Xinje XDPPro project, PLC1: XDH-60T4 (software 3.7.14b 2022-06-24)

PROGRAM 梯形图

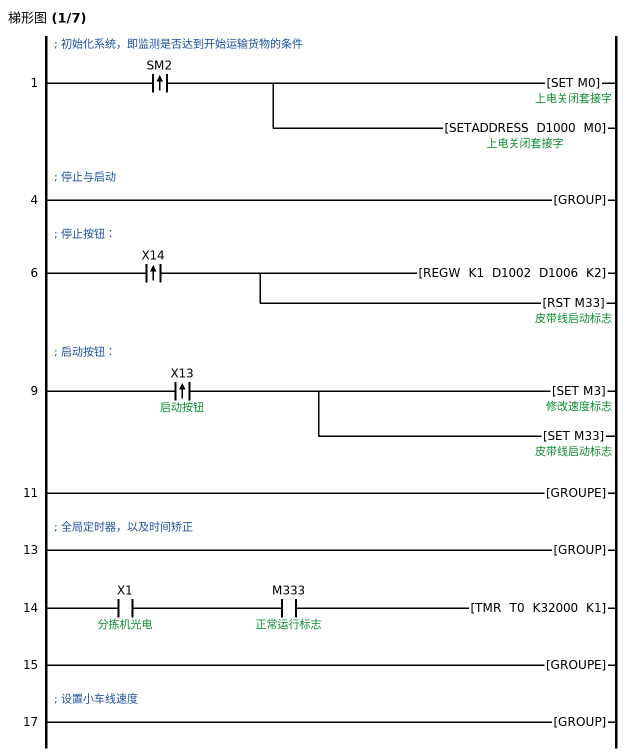
; 初始化系统，即监测是否达到开始运输货物的条件
LDP    SM2
SET    M0	; 上电关闭套接字
SETADDRESS D1000 M0	; 上电关闭套接字
; 停止与启动
GROUP
; 停止按钮：
LDP    X14
REGW   K1 D1002 D1006 K2
RST    M33	; 皮带线启动标志
; 启动按钮：
LDP    X13	; 启动按钮
SET    M3	; 修改速度标志
SET    M33	; 皮带线启动标志
GROUPE
; 全局定时器，以及时间矫正
GROUP
LD     X1	; 分拣机光电
AND    M333	; 正常运行标志
TMR    T0 K32000 K1
GROUPE
; 设置小车线速度
GROUP

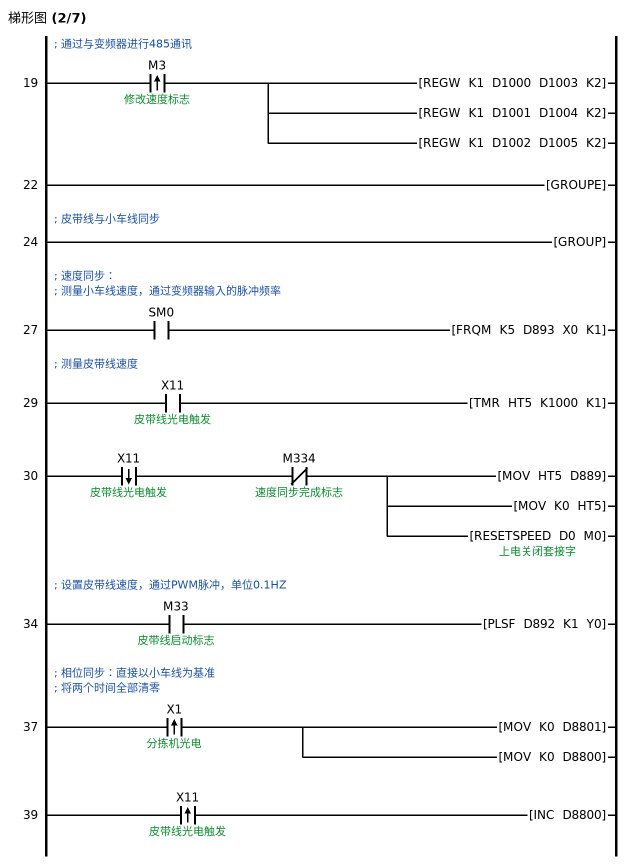
; 通过与变频器进行485通讯
LDP    M3	; 修改速度标志
REGW   K1 D1000 D1003 K2
REGW   K1 D1001 D1004 K2
REGW   K1 D1002 D1005 K2
GROUPE
; 皮带线与小车线同步
GROUP
; 速度同步：
; 测量小车线速度，通过变频器输入的脉冲频率
LD     SM0
FRQM   K5 D893 X0 K1
; 测量皮带线速度
LD     X11	; 皮带线光电触发
TMR    HT5 K1000 K1
LDF    X11	; 皮带线光电触发
ANI    M334	; 速度同步完成标志
MOV    HT5 D889
MOV    K0 HT5
RESETSPEED D0 M0	; 上电关闭套接字
; 设置皮带线速度，通过PWM脉冲，单位0.1HZ
LD     M33	; 皮带线启动标志
PLSF   D892 K1 Y0
; 相位同步：直接以小车线为基准
; 将两个时间全部清零
LDP    X1	; 分拣机光电
MOV    K0 D8801
MOV    K0 D8800
LDP    X11	; 皮带线光电触发
INC    D8800

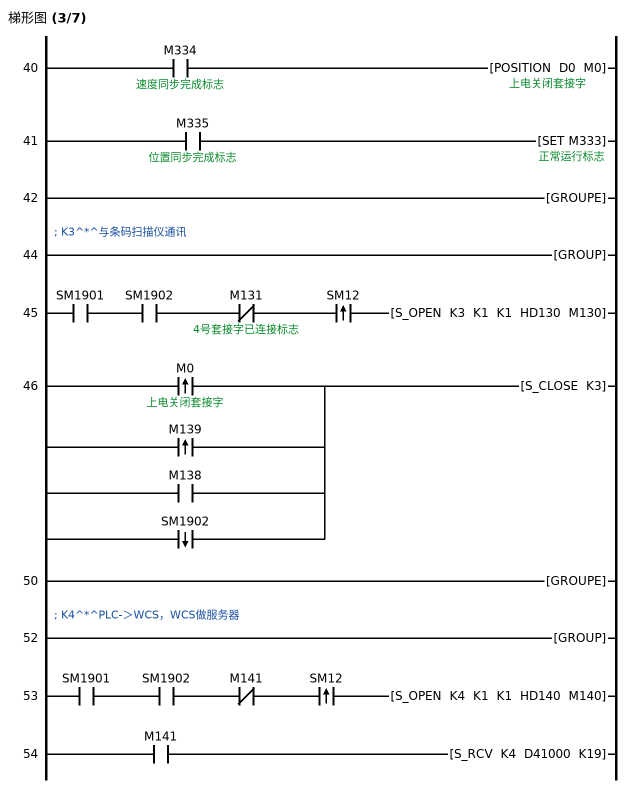
LD     M334	; 速度同步完成标志
POSITION D0 M0	; 上电关闭套接字
LD     M335	; 位置同步完成标志
SET    M333	; 正常运行标志
GROUPE
; K3^*^与条码扫描仪通讯
GROUP
LD     SM1901
AND    SM1902
ANI    M131	; 4号套接字已连接标志
ANDP   SM12
S_OPEN K3 K1 K1 HD130 M130
LDP    M0	; 上电关闭套接字
ORP    M139
OR     M138
ORF    SM1902
S_CLOSE K3
GROUPE
; K4^*^PLC-＞WCS，WCS做服务器
GROUP
LD     SM1901
AND    SM1902
ANI    M141
ANDP   SM12
S_OPEN K4 K1 K1 HD140 M140
LD     M141
S_RCV  K4 D41000 K19

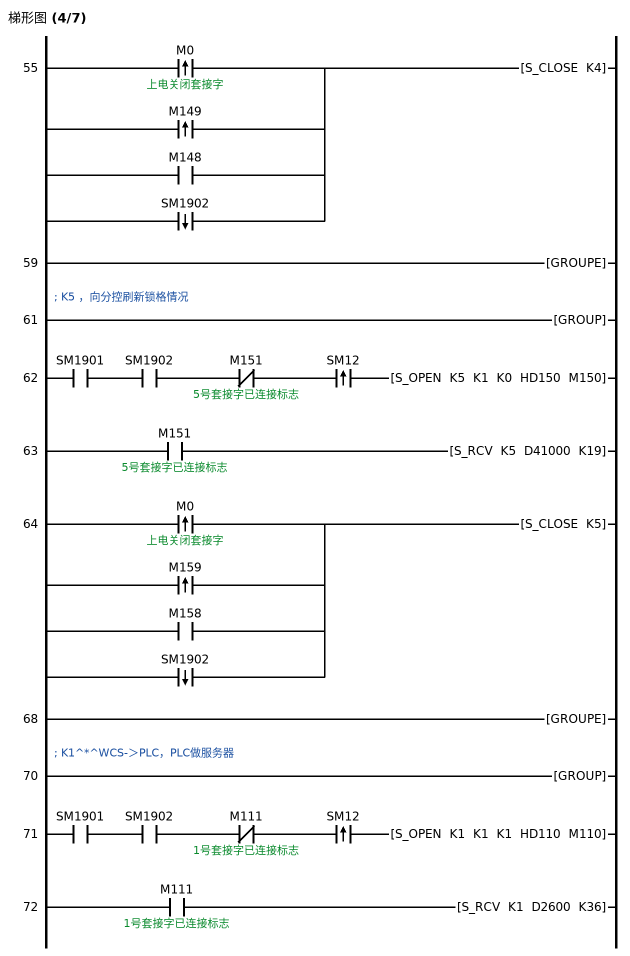
LDP    M0	; 上电关闭套接字
ORP    M149
OR     M148
ORF    SM1902
S_CLOSE K4
GROUPE
; K5 ，向分控刷新锁格情况
GROUP
LD     SM1901
AND    SM1902
ANI    M151	; 5号套接字已连接标志
ANDP   SM12
S_OPEN K5 K1 K0 HD150 M150
LD     M151	; 5号套接字已连接标志
S_RCV  K5 D41000 K19
LDP    M0	; 上电关闭套接字
ORP    M159
OR     M158
ORF    SM1902
S_CLOSE K5
GROUPE
; K1^*^WCS-＞PLC，PLC做服务器
GROUP
LD     SM1901
AND    SM1902
ANI    M111	; 1号套接字已连接标志
ANDP   SM12
S_OPEN K1 K1 K1 HD110 M110
LD     M111	; 1号套接字已连接标志
S_RCV  K1 D2600 K36

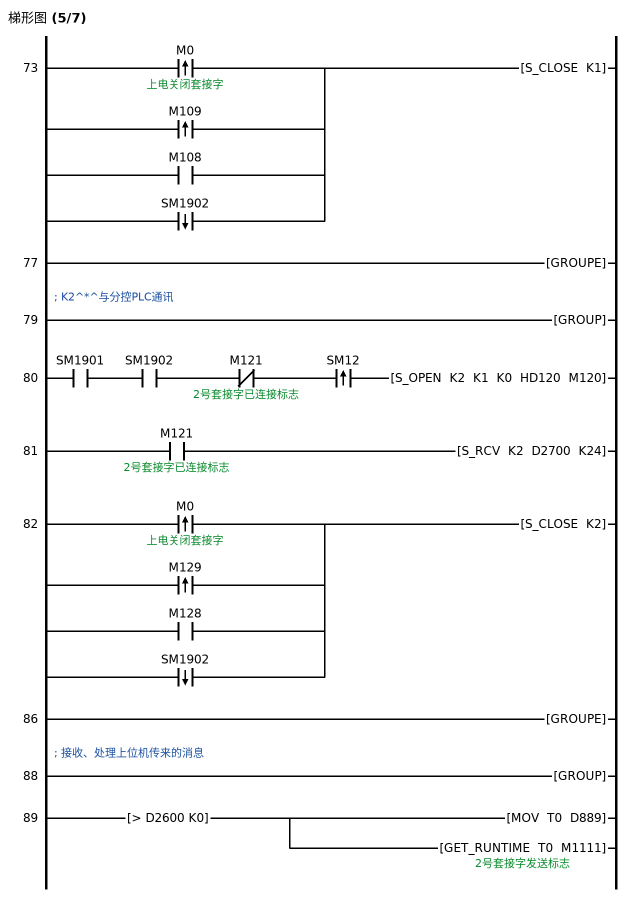
LDP    M0	; 上电关闭套接字
ORP    M109
OR     M108
ORF    SM1902
S_CLOSE K1
GROUPE
; K2^*^与分控PLC通讯
GROUP
LD     SM1901
AND    SM1902
ANI    M121	; 2号套接字已连接标志
ANDP   SM12
S_OPEN K2 K1 K0 HD120 M120
LD     M121	; 2号套接字已连接标志
S_RCV  K2 D2700 K24
LDP    M0	; 上电关闭套接字
ORP    M129
OR     M128
ORF    SM1902
S_CLOSE K2
GROUPE
; 接收、处理上位机传来的消息
GROUP
LD>    D2600 K0
MOV    T0 D889
GET_RUNTIME T0 M1111	; 2号套接字发送标志

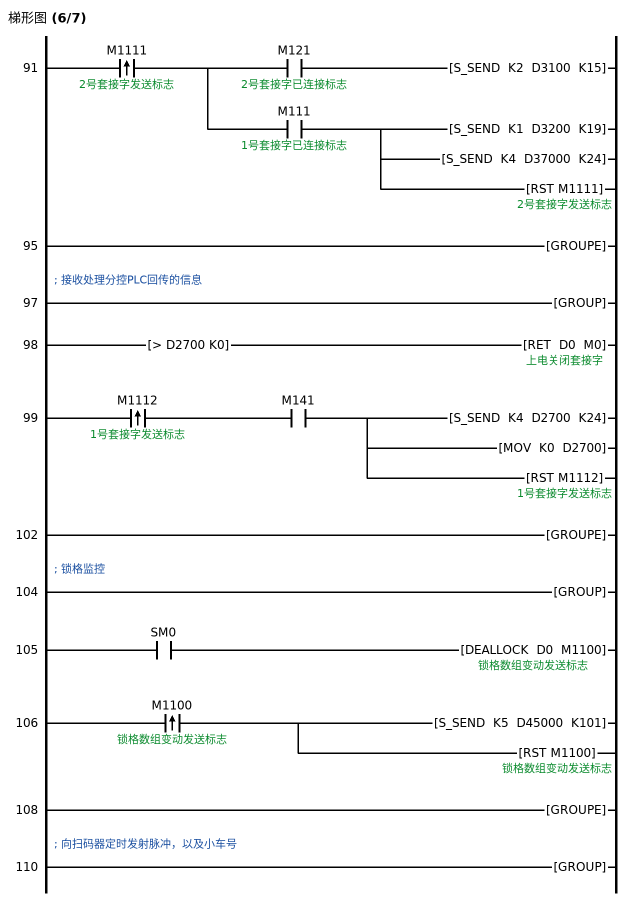
LDP    M1111	; 2号套接字发送标志
MPS
AND    M121	; 2号套接字已连接标志
S_SEND K2 D3100 K15
MPP
AND    M111	; 1号套接字已连接标志
S_SEND K1 D3200 K19
S_SEND K4 D37000 K24
RST    M1111	; 2号套接字发送标志
GROUPE
; 接收处理分控PLC回传的信息
GROUP
LD>    D2700 K0
RET    D0 M0	; 上电关闭套接字
LDP    M1112	; 1号套接字发送标志
AND    M141
S_SEND K4 D2700 K24
MOV    K0 D2700
RST    M1112	; 1号套接字发送标志
GROUPE
; 锁格监控
GROUP
LD     SM0
DEALLOCK D0 M1100	; 锁格数组变动发送标志
LDP    M1100	; 锁格数组变动发送标志
S_SEND K5 D45000 K101
RST    M1100	; 锁格数组变动发送标志
GROUPE
; 向扫码器定时发射脉冲，以及小车号
GROUP

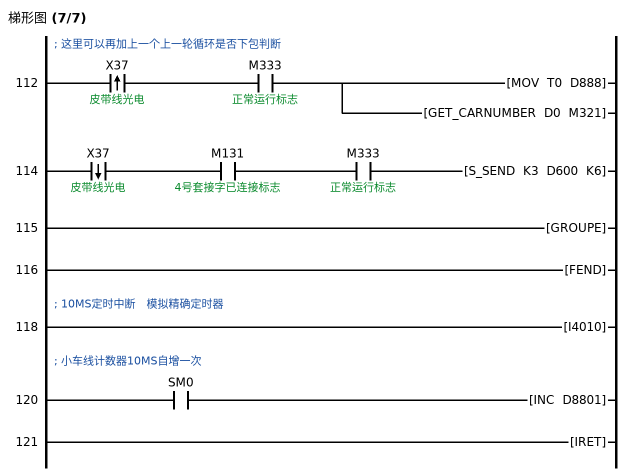
; 这里可以再加上一个上一轮循环是否下包判断
LDP    X37	; 皮带线光电
AND    M333	; 正常运行标志
MOV    T0 D888
GET_CARNUMBER D0 M321
LDF    X37	; 皮带线光电
AND    M131	; 4号套接字已连接标志
AND    M333	; 正常运行标志
S_SEND K3 D600 K6
GROUPE
FEND
; 10MS定时中断　模拟精确定时器
I4010
; 小车线计数器10MS自增一次
LD     SM0
INC    D8801
IRET

COMMENTS (devices not used above)
M101	1号套接字已连接
M99	3号套接字发送标志
HD10	定时器最大值
HD11	定时器数量
Y1	控制伺服电机方向

C FUNCTION BLOCK deallock.fcb
/* 处理、检测锁格的情况
#EXPORT_ENTRY_BEGIN(DEALLOCK)
//    类型              模式             个数               映射          注释
W = { type = "PINT16S", mode = [In,Out], count = "unknown", map = [D,HD], comment = "" }
B = { type = "BIT"    , mode = [In,Out], count = "unknown", map = [M,HM], comment = "" }
#EXPORT_ENTRY_END */
/*************************************************************************
 * FunctionBlockName:  DEALLOCK
 * Version:            1.0.0
 * Author:             rpl
 * UpdateTime:         2022-09-13 14:35:26
 * Comment:            处理、检测锁格的情况
**************************************************************************/

/**
 * @summary 
 * @param W 
 * @param B 
 */
 
 #include"func1.h"

void DEALLOCK(PINT16S W,BIT B)
{
	#define SysRegAddr_HD_D_HM_M_X_Y
	
    *(LOCKFIRSTADDRESS) = 0x02;
	for(int i = 30; i<=SIZEOFLATTICE;i++)
    {
    	if(X[i]!= *(LOCKFIRSTADDRESS+i+1))
        {
                //发送位置1
                M[1100] = 1;
        }
        * ( LOCKFIRSTADDRESS + i+1 ) = X[i];
    }
    return;
}

C FUNCTION BLOCK dealwith_k1.fcb
/* #EXPORT_ENTRY_BEGIN(DEALWITH_K1)
//    类型              模式             个数               映射          注释
W = { type = "PINT16S", mode = [In,Out], count = "unknown", map = [D,HD], comment = "" }
B = { type = "BIT"    , mode = [In,Out], count = "unknown", map = [M,HM], comment = "" }
#EXPORT_ENTRY_END */
/*************************************************************************
 * FunctionBlockName:  DEALWITH_K1
 * Version:            1.0.0
 * Author:             
 * UpdateTime:         2022-08-22 14:10:12
 * Comment:            
**************************************************************************/

/**
 * @summary 
 * @param W 
 * @param B 
 */
void DEALWITH_K1(PINT16S W,BIT B)
{
	#define SysRegAddr_HD_D_HM_M
    M[103] = 0;
    M[1112]　 = 0;

}

C FUNCTION BLOCK dealwith_k2.fcb
/* #EXPORT_ENTRY_BEGIN(DEALWITH_K2)
//    类型              模式             个数               映射          注释
W = { type = "PINT16S", mode = [In,Out], count = "unknown", map = [D,HD], comment = "" }
B = { type = "BIT"    , mode = [In,Out], count = "unknown", map = [M,HM], comment = "" }
#EXPORT_ENTRY_END */
/*************************************************************************
 * FunctionBlockName:  DEALWITH_K2
 * Version:            1.0.0
 * Author:             
 * UpdateTime:         2022-08-22 14:08:06
 * Comment:            
**************************************************************************/

/**
 * @summary 
 * @param W 
 * @param B 
 */
void DEALWITH_K2(PINT16S W,BIT B)
{
	#define SysRegAddr_HD_D_HM_M
    M[113] = 0;
    M[1111] = 0;

}

C FUNCTION BLOCK func1.fcb
/* #EXPORT_ENTRY_BEGIN(FUNC1)
//    类型              模式             个数               映射          注释
W = { type = "PINT16S", mode = [In,Out], count = "unknown", map = [D,HD], comment = "" }
B = { type = "BIT"    , mode = [In,Out], count = "unknown", map = [M,HM], comment = "" }
#EXPORT_ENTRY_END */
/*************************************************************************
 * FunctionBlockName:  FUNC1
 * Version:            1.0.0
 * Author:             
 * UpdateTime:         2022-08-18 08:24:01
 * Comment:            
**************************************************************************/

/**
 * @summary 
 * @param W 
 * @param B 
 */
void FUNC1(PINT16S W,BIT B)
{
	#define SysRegAddr_HD_D_HM_M

}

C FUNCTION BLOCK get_carnumber.fcb
/* 输入时间，返回当前相机拍摄的小车号
#EXPORT_ENTRY_BEGIN(GET_CARNUMBER)
//    类型              模式             个数               映射          注释
W = { type = "PINT16S", mode = [In,Out], count = "unknown", map = [D,HD], comment = "" }
B = { type = "BIT"    , mode = [In,Out], count = "unknown", map = [M,HM], comment = "" }
#EXPORT_ENTRY_END */
/*************************************************************************
 * FunctionBlockName:  GET_CARNUMBER
 * Version:            1.0.0
 * Author:             rpl
 * UpdateTime:         2022-08-10 14:44:36
 * Comment:            输入时间,返回当前相机拍摄的小车号,将返回数据处理发给扫码仪
**************************************************************************/

/**
 * @summary
 * @param W
 * @param B
 */
#include"func1.h"


void GET_CARNUMBER ( PINT16S W, BIT B )
{
#define SysRegAddr_HD_D_HM_M_T
    /*根据时间判断出当前是多少号小车(小车从0号开始排序) */
    INT32U tmpp =  Speed * PassedTime*10;
    INT16U carnumber;
    if(tmpp >= Light2CameraPosition)
    {
        carnumber = ( (tmpp -Light2CameraPosition) / DistanceOfCar ) + 1;  //判断是哪个小车,用来绑定小车的控制电机计时时间
    }
    else{
        carnumber = ( (tmpp + Camera_Position)/ DistanceOfCar ) + 1;  //判断是哪个小车,用来绑定小车的控制电机计时时间
        
    }
    



    /***将小车号数据写入寄存器,起始位置D600,6个***/
    //消息头
    //int TempCar = carnumber;
    * ( SendToCameraFirstAddress ) = 0x02;
    //千位
    * ( SendToCameraFirstAddress + 1 ) = 0x30;
    //百位
    * ( SendToCameraFirstAddress + 2 ) = 48 + ( carnumber / 100 ) % 10 ;
    //十位
    * ( SendToCameraFirstAddress + 3 ) = 48 + ( carnumber / 10 ) % 10;
    //个位
    * ( SendToCameraFirstAddress + 4 ) = 48 + carnumber % 10;
    //结束符
    * ( SendToCameraFirstAddress + 5 ) = 0x03;



    //M[321] = 1;
    return;
}

C FUNCTION BLOCK get_runtime.fcb
/* D[100]返回某个电机在多少秒后运行,D[101]返回判断出的小车号，以此来进行绑定
#EXPORT_ENTRY_BEGIN(GET_RUNTIME)
//    类型          模式             个数               映射          注释
w = { type = "BIT", mode = [In]    , count = "1"      , map = [T]   , comment = "时间差" }
B = { type = "BIT", mode = [In,Out], count = "unknown", map = [M,HM], comment = ""    }
#EXPORT_ENTRY_END */
/*************************************************************************
 * FunctionBlockName:  GET_RUNTIME
 * Version:            1.0.0
 * Author:             rpl
 * UpdateTime:         2022-07-25 16:38:06
 * Comment:            处理上位机发来的数据，返回的ACK报文，写入发送缓冲区，
**************************************************************************/

/**
 * @summary
 * @param w 时间差
 * @param B
 */
#include "func1.h"

void GET_RUNTIME ( BIT w, BIT B )
{
#define SysRegAddr_HD_D_HM_M_T
    /** 分拣指令	0x02(起始符(16进制))	1(报文类型ASCII)
        齐格控制	0x02(起始符(16进制))	2(报文类型ASCII)
        锁格控制	0x02(起始符(16进制))	3(报文类型ASCII)
    */


    int master = * ( RCVDateFirstAddress + 1 );
    switch ( master )
    {
        case 49:
        {
            /**先处理接受到的报文,得到其中的小车号,格口号**/
            //先处理小车号码
            INT16U Car_Mark ;
            Car_Mark = ( *(RCVDateFirstAddress+10) - 48 ) * 1000 + ( *(RCVDateFirstAddress+11) - 48 ) * 100 + ( *(RCVDateFirstAddress+12) - 48 ) * 10 + *(RCVDateFirstAddress+13) - 48 ;
            
            INT16U Bourn1, Bourn2, Bourn3, Bourn4;
            INT16U  NeedTime1, NeedTime2, NeedTime3, NeedTime4;
            //如果小车号为0,即为返回报文 ,暂时不作处理直接丢弃
            if ( Car_Mark == 0 )
            {
                return;
            }
            //处理格口号
            Bourn1 = ( *(RCVDateFirstAddress+14) - 48 ) * 1000 + ( *(RCVDateFirstAddress+15) - 48 ) * 100 + ( *(RCVDateFirstAddress+16) - 48 ) * 10 + *(RCVDateFirstAddress+17) - 48 ;
            Bourn2 = ( *(RCVDateFirstAddress+18) - 48 ) * 1000 + ( *(RCVDateFirstAddress+19) - 48 ) * 100 + ( *(RCVDateFirstAddress+20) - 48 ) * 10 + *(RCVDateFirstAddress+21) - 48 ;
            Bourn3 = ( *(RCVDateFirstAddress+22) - 48 ) * 1000 + ( *(RCVDateFirstAddress+23) - 48 ) * 100 + ( *(RCVDateFirstAddress+24) - 48 ) * 10 + *(RCVDateFirstAddress+25) - 48 ;
            Bourn4 = ( *(RCVDateFirstAddress+26) - 48 ) * 1000 + ( *(RCVDateFirstAddress+27) - 48 ) * 100 + ( *(RCVDateFirstAddress+28) - 48 ) * 10 + *(RCVDateFirstAddress+29) - 48 ;
            INT16U time = D[889] * 10;
            NeedTime1 = ( Bourn1 * DistanceOfCut + ( Car_Mark - 1 ) * DistanceOfCar ) / Speed  - time; //总时间减去已经用的时间
            NeedTime2 = ( Bourn2 * DistanceOfCut + ( Car_Mark - 1 ) * DistanceOfCar ) / Speed  - time;
            NeedTime3 = ( Bourn3 * DistanceOfCut + ( Car_Mark - 1 ) * DistanceOfCar ) / Speed  - time;
            NeedTime4 = ( Bourn4 * DistanceOfCut + ( Car_Mark - 1 ) * DistanceOfCar ) / Speed  - time;
            //}
            
            //将数据填入发送缓冲区
            //首位
            * ( SendToLowPLCBuffAddress ) = 0x02;
            //定时1
            * ( SendToLowPLCBuffAddress + 1 ) = NeedTime1 >> 8;
            * ( SendToLowPLCBuffAddress + 2 ) = ( NeedTime1 << 8 ) >> 8;
            //定时2
            * ( SendToLowPLCBuffAddress + 3 ) = NeedTime2 >> 8;
            * ( SendToLowPLCBuffAddress + 4 ) = ( NeedTime2 << 8 ) >> 8;
            //定时3
            * ( SendToLowPLCBuffAddress + 5 ) = NeedTime3 >> 8;
            * ( SendToLowPLCBuffAddress + 6 ) = ( NeedTime3 << 8 ) >> 8;
            //定时四
            * ( SendToLowPLCBuffAddress + 7 ) = NeedTime4 >> 8;
            * ( SendToLowPLCBuffAddress + 8 ) = ( NeedTime4 << 8 ) >> 8;
            //格口
            
            //格口1
            * ( SendToLowPLCBuffAddress + 9 ) = Bourn1;
            //格口2
            * ( SendToLowPLCBuffAddress + 10 ) = Bourn2;
            //格口3
            * ( SendToLowPLCBuffAddress + 11 ) = Bourn3;
            //格口4
            * ( SendToLowPLCBuffAddress + 12 ) = Bourn4;
            //小车号
            * ( SendToLowPLCBuffAddress + 13 ) = Car_Mark;
            //命令语
            * ( SendToLowPLCBuffAddress + 14 ) = master;
            break;
        }
        case 50: //齐格指令
        break;
        case 51://锁格指令
        break;
    }
    
    
    



    /**************************************处理向上位机回复ACK信息************************
     1.起始位置D3200               ***
     2.发送19个寄存器的数据        ***
     *************/
     *(SendACKToWCSFiestAddress) = 0x02;

    /**将报文编号复制到1号套接字发送缓冲区*/
    for ( int i = 1; i <= 8; i++ )
    {
        *(SendACKToWCSFiestAddress +i) = *(RCVDateFirstAddress+1+i);
    }
    for ( int i = 9; i <= 12; i++ )
    {
        *(SendACKToWCSFiestAddress +i)  = 48;
    }

    for ( int i = 13; i <= 17; i++ )
    {
        *(SendACKToWCSFiestAddress +i) = 0x20;
    }
    //结束符
    *(SendACKToWCSFiestAddress +18) = 0x03;

    //将接受区的数据清零
    *(RCVDateFirstAddress) = 0;
    //出发发送数据用
    M[1111] = 1;
    return;
}

C FILE func1.h
#ifndef	_FUNC1_H
#define	_FUNC1_H
/*********宏定义用来存放需要的返回值************/
 //#define NEEDTIME D[3100]       //保存返回值
 //#define CAR      D[3102]        //存储判断出来的小车号
 //#define Bourn     D[3103]       //目的格口
 //#define Time      D[300]           //时间基点定时器的计数值 
#define D_D	     *(INT32S*)&D


/**********首地址************/
#define SendToLowPLCBuffAddress D+3100 //发送给分控的发送缓冲区首地址,总计15个寄存器
#define RCVDateFirstAddress D+2600      //上位机发来的数据缓冲区首地址，总计36个寄存器
#define SendACKToWCSFiestAddress D+3200 //向上位机回复ACK报文的数据缓冲区首地址，总计19个寄存器
#define SendToCameraFirstAddress D+600  //发给相机，6个寄存器
#define RCVDateFormLOW          D+2700  //分控分拣完成返回，24个寄存器
#define LOCKFIRSTADDRESS D+45000        //锁格队列首地址,101个寄存器
#define CarDateFirstAddress D+3300      //存放已有任务的小车数组


/* 存放一些函数中需要的参数 
所有的距离单位为毫米，时间单位为毫秒
 */
 
 
 #define TrackLength  50000         //轨道的长度
 #define  Speed  1                  //小车速度1mm/ms
 #define DistanceOfCar  400         //小车的间距(单位为：毫米)
 #define TIMELOSS  5                //电机启动时间偏移量(单位为：毫秒)

 #define Time_Offset 　0            //时间偏移量，由于没有进行实验测试暂时设置为0,该值是用来计算小车上的电机转动所需要的时间

 #define DistanceOfCut  750         //此处割口的间距 ————割口的长度加上割口间的距离

 #define  Camera_Position  600      //扫码设备->光电的距离
 #define Light2CameraPosition (TrackLength-Camera_Position)  //光电->扫码设备的距离

 #define Time  0                    //距离时间基点的时间

 
 #define SIZEOFLATTICE 100      //格口个数


//小车线与皮带线用
#define PassedTime      D[888]
#define NowSpeed        D[890]         //皮带线当前速度
#define CarSpeed        D[891]         //小车线速度
#define PulseFrequency  D[892]   //皮带线脉冲频率
#define FinallyFrequency  D[894]    //皮带线最终脉冲频率
#define CarFrequency    D[893]   //小车线反馈脉冲频率
#define speedAddress     D[1000]  //Modbus转速地址
#define PowerAddress     D[1001]  //转矩地址
#define MasterAddress    D[1002]  //命令符地址
#define speedValue       D[1003]  //转速数值
#define PowerValue       D[1004]  //转矩数值
#define MasterValue      D[1005]  //命令符
#define StopMaster       D[1006]    //电机停止
#define CarIncConter   D[8801]  //小车线当前时间
#define PulseIncConter D[8800]  //皮带线当前计数值

#define CameraEnableTime D[894]     //相机使能定时时间
#define DZCL        D[8802]     //转一圈需要的脉冲数

#endif

C FUNCTION BLOCK init.fcb
/* 初始化需要的数组，结构体
#EXPORT_ENTRY_BEGIN(INIT)
//    类型              模式             个数               映射          注释
W = { type = "PINT16S", mode = [In,Out], count = "unknown", map = [D,HD], comment = "" }
B = { type = "BIT"    , mode = [In,Out], count = "unknown", map = [M,HM], comment = "" }
#EXPORT_ENTRY_END */
/*************************************************************************
 * FunctionBlockName:  INIT
 * Version:            1.0.0
 * Author:             rpl
 * UpdateTime:         2022-09-13 15:01:51
 * Comment:            初始化需要的数组，结构体
**************************************************************************/

/**
 * @summary 
 * @param W 
 * @param B 
 */
 #include"func1.h"
void INIT(PINT16S W,BIT B)
{
	#define SysRegAddr_HD_D_HM_M
	for(int i = 0;i<=SIZEOFLATTICE; i++)
    {
        * ( LOCKFIRSTADDRESS + i ) = 0;
    }
	
	

}

C FUNCTION BLOCK position.fcb
/* 位置矫正，皮带线与分拣机的相位矫正。
#EXPORT_ENTRY_BEGIN(POSITION)
//    类型              模式             个数               映射          注释
W = { type = "PINT16S", mode = [In,Out], count = "unknown", map = [D,HD], comment = "" }
B = { type = "BIT"    , mode = [In,Out], count = "unknown", map = [M,HM], comment = "" }
#EXPORT_ENTRY_END */
/*************************************************************************
 * FunctionBlockName:  POSITION
 * Version:            1.0.0
 * Author:             rpl
 * UpdateTime:         2022-09-28 16:15:44
 * Comment:            位置矫正，皮带线与分拣机的相位矫正。
                        这里默认已经进行过基本的速度矫正
**************************************************************************/

/**
 * @summary 
 * @param W 
 * @param B 
 */
 #include"func1.h"
void POSITION(PINT16S W,BIT B)
{
	#define SysRegAddr_HD_D_HM_M
    /*需要做的事情
    1.两条线的计数器时间之差： 分拣机的可以通过时间进行自增 保持精度与皮带线相同或者大十倍
    2.频率对应的关系变量
    3.微调是通过固定值加减还是通过速度公式去追及，在追及的时候速度什么时候降到与分拣机相同，在下一次的光电信号到来之前是无法判断当前相位差的
    4.速度与频率关系的对应公式！！！
    */
    /*新增控制部分需要的参数 
    1.直线电机的运行速度 V    1.0 mm/ms  1.0 m/s
    2.伺服电机的电子齿轮比 K 10000:10000  
    3.伺服电机旋转一圈的长度 C   440 mm    
    4.脉冲：距离 = 10000 ： 500
    5.脉冲频率 H
    6. 伺服电机速度（单位 mm/s） =
    
    7. 伺服电机当前频率 PulseFrequency
    8.两条线的计数值之差 CounterDifference
    9.单位步进值  UnitStepValue
    */
    //int CarIncCounter; //乘以10等于小车线当前走的时间
    //int PulseFrequency;     //间距除以速度等于皮带线当前走的时间
    //int UnitStepValue =  DZCL*10 *DistanceOfCar / 0.44;
    int CarDistance  =  CarIncCounter * 10 * Speed; //单位ms
    int BeltDistance =  PulseIncConter * DistanceOfCar; // 单位mm
    int DistanceDifference = CarDistance - BeltDistance; //两条线的相位差
    /**拟通过单位步进值来进行处理，但应该是行不通的*/
    /*每次增加1000个脉冲——0.1375m/s的速度去追及*/
    if(DistanceDifference >=0)
    { 
        PulseFrequency += 1000 ;
    }
    else if(DistanceDifference < 0)
    {
        PulseFrequency -= 1000; 
    }

    //相位矫正完成
    if(DistanceDifference >= -10 || DistanceDifference <= 10 )
    {
        //将速度重置为最终速度
        PulseFrequency = FinallyFrequency;
        
        M[335] = 1;     //相位同步完成标志
    }
    else
    {
    M[335] = 0;
    }

return;
}

C FUNCTION BLOCK resetspeed.fcb
/* 皮带线速度向小车线靠近
#EXPORT_ENTRY_BEGIN(RESETSPEED)
//    类型              模式             个数               映射          注释
W = { type = "PINT16S", mode = [In,Out], count = "unknown", map = [D,HD], comment = "" }
B = { type = "BIT"    , mode = [In,Out], count = "unknown", map = [M,HM], comment = "" }
#EXPORT_ENTRY_END */
/*************************************************************************
 * FunctionBlockName:  RESETSPEED
 * Version:            1.0.0
 * Author:             
 * UpdateTime:         2022-10-06 17:14:06
 * Comment:            皮带线速度向小车线靠近
**************************************************************************/

/**
 * @summary 
 * @param W 
 * @param B 
 */
 #include"func1.h"
 #define TimeValue D[889]
void RESETSPEED(PINT16S W,BIT B)
{
	#define SysRegAddr_HD_D_HM_M
    float deviation = 0.05; //允许误差
    NowSpeed =  DistanceOfCar / TimeValue;//单位 mm/ms
    CarSpeed = CarFrequency * 0.1; //单位m/s
    if (NowSpeed < CarSpeed)
    { 
        //此处假设1000个脉冲转一圈
        PulseFrequency = PulseFrequency + ( ( CarSpeed - NowSpeed ) *1000/137.5);
        //百分比*额度转速*减速比 = 实际转速
        //实际转速*0.44 = 线速度
        //调整后的频率= 当前频率+差值速度*100000  /0.44/减速比/额定转速
    }
    else if(NowSpeed > CarSpeed)
    {
        PulseFrequency = PulseFrequency - ( ( NowSpeed -CarSpeed) *1000/137.5);
    }
    //脉冲乘以减速比
    PulseFrequency = PulseFrequency * 16;
	//当速度达到允许误差时，速度同步完成标志置1
	if(NowSpeed == CarSpeed || NowSpeed - CarSpeed <=deviation ||  CarSpeed - NowSpeed <=deviation )
	{
	    //保存速度同步完成的频率
        PulseFrequency = FinallyFrequency;
        M[334] = 1;
	}
	////超过最大允许误差时，将速度同步完成标志置0
	//else
	//{
	    
	    //M[334] = 0;
	//}
    return;
}

C FUNCTION BLOCK ret.fcb
/* 向上位机返回ack
#EXPORT_ENTRY_BEGIN(RET)
//    类型              模式             个数               映射          注释
W = { type = "PINT16S", mode = [In,Out], count = "unknown", map = [D,HD], comment = "" }
B = { type = "BIT"    , mode = [In,Out], count = "unknown", map = [M,HM], comment = "" }
#EXPORT_ENTRY_END */
/*************************************************************************
 * FunctionBlockName:  RET
 * Version:            1.0.0
 * Author:             
 * UpdateTime:         2022-09-08 15:23:59
 * Comment:            向上位机返回ack
**************************************************************************/

/**
 * @summary 
 * @param W 
 * @param B 
 */
 #define SendToWCSFirstAddress D+37000
 #include"func1.h"
void RET(PINT16S W,BIT B)
{
	#define SysRegAddr_HD_D_HM_M
	//落格成功返回
	
	//起始符
    *(SendToWCSFirstAddress) = 0x02;
    //分拣完成
    *(SendToWCSFirstAddress+1) = 53;
    
    //报文编号
    for(int i = 2; i<=9;i++)
    {
        *(SendToWCSFirstAddress+i) = *(RCVDateFormLOW+i);
    }
    //小车号
    for(int i =10;i<=13; i++)
    {
        *(SendToWCSFirstAddress+i) = *(RCVDateFormLOW+i);
    }
    //格口
    for(int i=14;i<=16;i++)
    {
       *(SendToWCSFirstAddress+i) = *(RCVDateFormLOW+i);
    }
    //五位空格
    for(int i =17;i<=21;i++)
    {
        *(SendToWCSFirstAddress+i) = 32;
    }
   *(SendToWCSFirstAddress+23) = 0x03;
   
   * ( RCVDateFormLOW ) = 0; //接收区首地址置0 
}

C FUNCTION BLOCK setaddress.fcb
/* #EXPORT_ENTRY_BEGIN(SETADDRESS)
//    类型              模式             个数               映射          注释
W = { type = "PINT16S", mode = [In,Out], count = "unknown", map = [D,HD], comment = "" }
B = { type = "BIT"    , mode = [In,Out], count = "unknown", map = [M,HM], comment = "" }
#EXPORT_ENTRY_END */
/*************************************************************************
 * FunctionBlockName:  SETADDRESS
 * Version:            1.0.0
 * Author:             rpl
 * UpdateTime:         2022-08-25 16:03:02
 * Comment:            
**************************************************************************/

/**
 * @summary 
 * @param W 
 * @param B 
 */
 #include"func1.h"
void SETADDRESS(PINT16S W,BIT B)
{
	#define SysRegAddr_HD_D_HM_M
    speedAddress = 0x7002;
    PowerAddress = 0x7006;
    MasterAddress = 0x7000;
    speedValue  = 1000;
    PowerValue  = 1000;
    MasterValue = 0x0001;
    StopMaster = 0x0110;
    PulseFrequency =speedValue/1.375*10;
}

C FUNCTION BLOCK sub_control_return.fcb
/* 处理分控回传的数据
#EXPORT_ENTRY_BEGIN(SUB_CONTROL_RETURN)
//    类型              模式             个数               映射          注释
W = { type = "PINT16S", mode = [In,Out], count = "unknown", map = [D,HD], comment = "" }
B = { type = "BIT"    , mode = [In,Out], count = "unknown", map = [M,HM], comment = "" }
#EXPORT_ENTRY_END */
/*************************************************************************
 * FunctionBlockName:  SUB_CONTROL_RETURN
 * Version:            1.0.0
 * Author:             rpl
 * UpdateTime:         2022-08-19 10:53:12
 * Comment:            处理分控回传的数据
**************************************************************************/

/**
 * @summary 
 * @param W 
 * @param B 
 */
 
 
 /**分控plc回传的数据存放的首地址在D2700**/
 /**************
 D2700   唯一标识符
 D2701   小车号
 D2702   格口号


 ****************/
void SUB_CONTROL_RETURN(PINT16S W,BIT B)
{
    #define SysRegAddr_HD_D_HM_M


    
    
    //置位上升沿触发开关
    M[1112] = 1;
    
    
}